FUNCTION_BLOCK counter (* Basic Function Block Type *)
  (* Standard: 61499-2 *)
  (* Version 0.0, 5/24/2016, gulzha, nxtControl GmbH, Template *)
  PACKAGE Main;
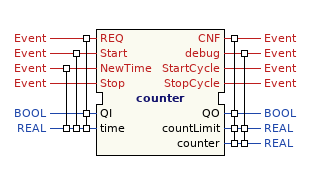
  EVENT_INPUT
    REQ WITH QI, time; (* Normal Execution Request *)
    Start WITH time;
    NewTime WITH time;
    Stop;
  END_EVENT
  EVENT_OUTPUT
    CNF WITH QO, countLimit, counter; (* Execution Confirmation *)
    debug WITH countLimit, counter;
    StartCycle;
    StopCycle;
  END_EVENT
  VAR_INPUT
    QI : BOOL; (* Input event qualifier *)
    time : REAL; (* in seconds *)
  END_VAR
  VAR_OUTPUT
    QO : BOOL; (* Output event qualifier *)
    countLimit : REAL;
    counter : REAL;
  END_VAR
  VAR
    step : BOOL := FALSE;
    countLimitInt : REAL;
    counterInt : REAL;
  END_VAR
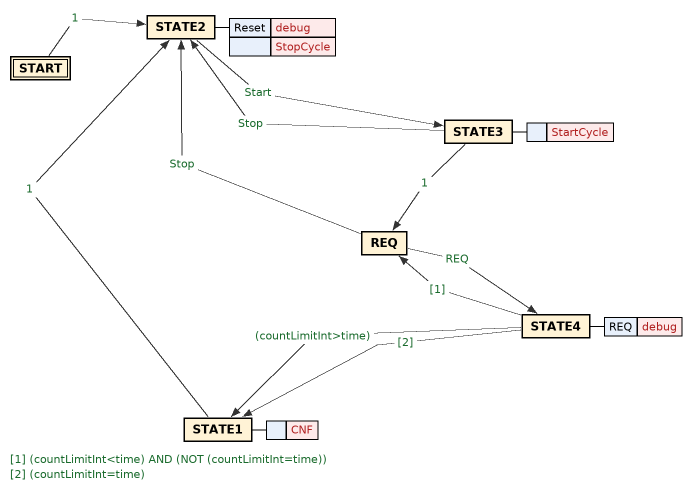
  EC_STATES
    START; (* Initial State *)
    REQ; (* Normal execution *)
    STATE1 : -> CNF;
    STATE2 : Reset -> debug, -> StopCycle;
    STATE3 : -> StartCycle;
    STATE4 : REQ -> debug;
  END_STATES
  EC_TRANSITIONS
    STATE4 TO STATE1 := (countLimitInt>time);
    STATE1 TO STATE2 := 1;
    START TO STATE2 := 1;
    STATE2 TO STATE3 := Start;
    REQ TO STATE2 := Stop;
    STATE3 TO STATE2 := Stop;
    REQ TO STATE4 := REQ;
    STATE4 TO REQ := (countLimitInt<time) AND (NOT (countLimitInt=time));
    STATE3 TO REQ := 1;
    STATE4 TO STATE1 := (countLimitInt=time);
  END_TRANSITIONS
  ALGORITHM REQ IN ST: (* Normally executed algorithm *)
;

//countLimit:= time/0.01;// divide the given time to 10 ms, result - counter limit
// e.g. 5 sec/ 0.01 = 500; count till 500 will give 5 seconds (interval 10 ms)
//countLimit:= time/0.005;
//countLimit:= time/0.005;
//countLimit:= time/0.001;
counterInt:=counterInt+1;
countLimitInt := counterInt * 0.002;


counter:=counterInt;
countLimit := countLimitInt;



//REQ:= FALSE;
  END_ALGORITHM
  ALGORITHM Reset IN ST:
;

countLimit:= 0;

counter:=0;
countLimitInt:= 0;

counterInt:=0;

step:=FALSE;
  END_ALGORITHM
END_FUNCTION_BLOCK
